Staubli VAL3: DeleteBuffTraj.pgx

public program DeleteBuffTraj()
  local num l_nNum
  local string l_sSFileName
begin

  //2015.04.24
  //为大数据文件报错

  for l_nNum=1 to 1000

    if $fileExists("Disk://Txt/"+toString("",l_nNum)+".txt")

      $delete("Disk://Txt/"+toString("",l_nNum)+".txt")
    else
      return
    endIf


  endFor





end
